// TIA Portal V20 export
VAR_GLOBAL   // PLC tag table "LGR_Const_System"
END_VAR
VAR_GLOBAL CONSTANT   // user constants
   TcpResQueMax : UInt := 255;
   EventQueMax : UInt := 255;
   CELL_ID_MAX : UInt := 1000;
   CELL_ID_MIN : UInt := 1;
   STATION_ID_MAX : UInt := 2999;
   STATION_ID_MIN : UInt := 2001;
   CELL_MIN : UInt := 1;
   STATION_MIN : UInt := 1;
   DebugLogMax : UInt := 19;
   PARA_MAX : UInt := 500;
   PARA_MIN : UInt := 1;
   PARA_NAME_MAX : UInt := 40;
   CSV_TYPE_PARA : UInt := 1;
   CSV_TYPE_CELL : UInt := 2;
   CSV_TYPE_STATION : UInt := 3;
   ZONE_ID_MIN : UInt := 1;
   ZONE_ID_MAX : UInt := 20;
   SAFETYZONE_MIN : UInt := 1;
   SAFETYZONE_MAX : UInt := 3;
   SCENARIO_MIN : UInt := 1;
   SCENARIO_MAX : UInt := 100;
   STATION_MAX : UInt := 32;
   CELL_MAX : UInt := 500;
   RIO_MODULE_COUNT : UInt := 2;
   IOLINK_MODULE_COUNT : UInt := 2;
   AXIS_MAX : UInt := 4;
   AXIS_MIN : UInt := 1;
   RESTRICTZONE_MIN : UInt := 1;
   RESTRICTZONE_MAX : UInt := 20;
   FENCEBOX_MIN : UInt := 1;
   FENCEBOX_MAX : UInt := 16;
   SAFETYDOOR_MIN : UInt := 1;
   SAFETYDOOR_MAX : UInt := 16;
   RIO_INPUT_COUNT : UInt := 13;
   RIO_OUTPUT_COUNT : UInt := 10;
END_VAR
